(* PLC project AutBoxInterfaceOpcUa_PW02_Solution.project, Rexroth ctrlX PLC Engineering ctrlX PLC 1.20.7 *)
(* stored: creationDateTime 2025-02-11T09:05:17.5730649, modificationDateTime 2024-03-01T13:41:48 *)

(* www.hevs.ch Institut Systemes Industriels Project: Projet No: PW_01 Author: Cedric Lenoir Date: 2023 October 11 Summary: List of of components for a station of a conveyor. *)
TYPE ST_StationConveyor : STRUCT
  bButton : BOOL;
  bLed : BOOL;
  bSensor : BOOL;
END_STRUCT;
END_TYPE

(* www.hevs.ch Institut Systemes Industriels Project: Projet No: PW_01 Author: Cedric Lenoir Date: 2023 October 11 Summary: List of of components for a motor of a conveyor. *)
TYPE ST_MotorConveyor : STRUCT
  bK_ActivatePositiveDirection : BOOL;
  bK_ActivateNegativeDirection : BOOL;
END_STRUCT;
END_TYPE

(* www.hevs.ch Institut Systemes Industriels Project: Projet No: PW_02 Author: Cedric Lenoir Date: 2024 January 16 Summary: Main structure for conveyor. *)
TYPE ST_Conveyor : STRUCT
  cm01 : ST_StationConveyor;
  cm02 : ST_StationConveyor;
  cm03 : ST_StationConveyor;
  cmOut : ST_OutputConveyor;
  cmDrive : ST_MotorConveyor;
END_STRUCT;
END_TYPE

(* www.hevs.ch Institut Systemes Industriels Project: Projet No: PW_01 Author: Cedric Lenoir Date: 2024 January 14 Summary: ST_OutputConveyor extends ST_StationConveyor. *)
TYPE ST_OutputConveyor : STRUCT
  bBuzzer : BOOL;
END_STRUCT;
END_TYPE

{attribute 'qualified_only'}
VAR_GLOBAL  (* GVL_Unit *)
  myConveyor : ST_Conveyor;
END_VAR

(* www.hevs.ch Institut Systemes Industriels Project: Projet No: PW_02 Author: Cedric Lenoir Date: 2024 January 16 Summary: Main program for Pracatival Work 02. *)
PROGRAM PLC_PRG
  VAR
    diMyLoop : DINT;
    emConveyor : ST_Conveyor;
    testMode : BOOL;
    fbStationOne : FB_Station;
    fbStationTwo : FB_Station;
    fbStationThree : FB_Station;
    fbOutStation : FB_OutStation;
    fbDrive : FB_Drive;
  END_VAR

            diMyLoop := diMyLoop + 1;

//
// Manage inputs
//
// cm01
emConveyor.cm01.bButton := GVL_Abox.uaAboxInterface.uaDigitalIn.Input_0_0;
emConveyor.cm01.bSensor := GVL_Abox.uaAboxInterface.uaDigitalIn.Input_0_4;	//  UA_DigitalInput_32_Input_0_4;
// cm02
emConveyor.cm02.bButton := GVL_Abox.uaAboxInterface.uaDigitalIn.Input_0_1;
emConveyor.cm02.bSensor := GVL_Abox.uaAboxInterface.uaDigitalIn.Input_0_5;
// cm03
emConveyor.cm03.bButton := GVL_Abox.uaAboxInterface.uaDigitalIn.Input_0_2;
emConveyor.cm03.bSensor := GVL_Abox.uaAboxInterface.uaDigitalIn.Input_0_6;
// cmOut
emConveyor.cmOut.bButton := GVL_Abox.uaAboxInterface.uaDigitalIn.Input_0_3;
emConveyor.cmOut.bSensor := NOT GVL_Abox.uaAboxInterface.uaDigitalIn.Input_0_7;	// Signal inverted

// To be tested
// FC_GetInput(ioHwInterface := GVL_Abox,
//             ioPhysicalControl := emConveyor);

fbStationOne(Enable := NOT testMode, 
          ioStation := emConveyor.cm01);
fbStationTwo(Enable := NOT testMode, 
          ioStation := emConveyor.cm02);
fbStationThree(Enable := NOT testMode, 
          ioStation := emConveyor.cm03);
		  
fbOutStation(Enable := NOT testMode, 
          ioStation := emConveyor.cmOut);

		  
fbDrive(Enable := NOT testMode,
		ioDrive := emConveyor.cmDrive,
        stationOne := fbStationOne,
        stationTwo := fbStationTwo,
        stationThree := fbStationThree,
        stationOut := fbOutStation);		  

//
// Manage outputs
//
// cm01
GVL_Abox.uaAboxInterface.uaDigitalOut.Output_0_0 := emConveyor.cm01.bLed;
GVL_Abox.uaAboxInterface.uaDigitalOut.Output_0_1 := emConveyor.cm02.bLed;
GVL_Abox.uaAboxInterface.uaDigitalOut.Output_0_2 := emConveyor.cm03.bLed;
GVL_Abox.uaAboxInterface.uaDigitalOut.Output_0_3 := emConveyor.cmOut.bLed;
GVL_Abox.uaAboxInterface.uaDigitalOut.Output_0_4 := emConveyor.cmDrive.bK_ActivatePositiveDirection;
GVL_Abox.uaAboxInterface.uaDigitalOut.Output_0_5 := emConveyor.cmDrive.bK_ActivateNegativeDirection;
GVL_Abox.uaAboxInterface.uaDigitalOut.Output_0_6 := emConveyor.cmOut.bBuzzer;

// To be tested
// FC_SetOutput(ioHwInterface := GVL_Abox,
//              ioPhysicalControl := emConveyor);
          
END_PROGRAM

(* www.hevs.ch Institut Systemes Industriels Project: Projet No: PW_02 Author: Cedric Lenoir Date: 2024 January 16 Summary: Manage One station for a conveyor. *)
FUNCTION_BLOCK FB_Station
  VAR_INPUT
    Enable : BOOL;
  END_VAR
  VAR_IN_OUT
    ioStation : ST_StationConveyor;
  END_VAR
  VAR_OUTPUT
    diCounter : DINT;
    stop : BOOL;
    release : BOOL;
  END_VAR
  VAR
    rTrigIn : R_TRIG;  (* Used to count the number of inputs in station *)
    tonResetCounter : TON;  (* Reset Counte if TON for more that 2 seconds *)
  END_VAR

            IF Enable THEN
	rTrigIn(CLK := ioStation.bSensor);
	
	IF rTrigIn.Q THEN
		diCounter := diCounter + 1;
		release := FALSE;
		stop := TRUE;
	END_IF
	IF ioStation.bButton THEN
		release := TRUE;
		stop := FALSE;
	END_IF
	ioStation.bLed := stop;
	
	tonResetCounter(IN := ioStation.bButton,
					PT := T#2S);
					
	IF tonResetCounter.Q THEN
		diCounter := 0;
	END_IF
END_IF
          
END_FUNCTION_BLOCK

(* www.hevs.ch Institut Systemes Industriels Project: Projet No: PW_02 Author: Cedric Lenoir Date: 2024 January 16 Summary: Manage One station for a conveyor. *)
FUNCTION_BLOCK FB_OutStation
  VAR_INPUT
    Enable : BOOL;
  END_VAR
  VAR_IN_OUT
    ioStation : ST_OutputConveyor;
  END_VAR
  VAR_OUTPUT
    diCounter : DINT;
    stop : BOOL;
    release : BOOL;
  END_VAR
  VAR
    rTrigIn : R_TRIG;  (* Used to count the number of inputs in station *)
    tonResetCounter : TON;  (* Reset Counte if TON for more that 2 seconds *)
  END_VAR

            IF Enable THEN
	rTrigIn(CLK := ioStation.bSensor);
	
	IF rTrigIn.Q THEN
		diCounter := diCounter + 1;
		release := FALSE;
		stop := TRUE;
	END_IF
	IF ioStation.bButton THEN
		release := TRUE;
		stop := FALSE;
	END_IF
	ioStation.bLed := stop;
	
	tonResetCounter(IN := ioStation.bButton,
					PT := T#2S);
					
	IF tonResetCounter.Q THEN
		diCounter := 0;
	END_IF
	
	ioStation.bBuzzer := stop;
END_IF
          
END_FUNCTION_BLOCK

(* www.hevs.ch Institut Systemes Industriels Project: Projet No: PW_02 Author: Cedric Lenoir Date: 2024 January 16 Summary: Manage drive for motor conveyor. *)
FUNCTION_BLOCK FB_Drive
  VAR_INPUT
    Enable : BOOL;
  END_VAR
  VAR_IN_OUT
    ioDrive : ST_MotorConveyor;
    stationOne : FB_Station;
    stationTwo : FB_Station;
    stationThree : FB_Station;
    stationOut : FB_OutStation;
  END_VAR

            IF Enable THEN
	ioDrive.bK_ActivatePositiveDirection := NOT(stationOne.stop   OR 
                                                stationTwo.stop   OR
                                                stationThree.stop OR
                                                stationOut.stop);
END_IF
          
END_FUNCTION_BLOCK

(* www.hevs.ch Institut Systemes Industriels Project: Projet No: PW_01 Author: Cedric Lenoir Date: 2023 October 11 Summary: Get Physical Inputs. *)
FUNCTION FC_GetInput : BOOL
  VAR_IN_OUT
    ioHwInterface : UA_AboxInterface;
    ioPhysicalControl : ST_Conveyor;
  END_VAR

            //
// Manage inputs
//
// cm01
ioPhysicalControl.cm01.bButton := ioHwInterface.uaDigitalIn.Input_0_0;
ioPhysicalControl.cm01.bSensor := ioHwInterface.uaDigitalIn.Input_0_4;	//  UA_DigitalInput_32_Input_0_4;
// cm02
ioPhysicalControl.cm02.bButton := ioHwInterface.uaDigitalIn.Input_0_1;
ioPhysicalControl.cm02.bSensor := ioHwInterface.uaDigitalIn.Input_0_5;
// cm03
ioPhysicalControl.cm03.bButton := ioHwInterface.uaDigitalIn.Input_0_2;
ioPhysicalControl.cm03.bSensor := ioHwInterface.uaDigitalIn.Input_0_6;
// cmOut
ioPhysicalControl.cmOut.bButton := ioHwInterface.uaDigitalIn.Input_0_3;
ioPhysicalControl.cmOut.bSensor := NOT ioHwInterface.uaDigitalIn.Input_0_7;	// Signal inverted
          
END_FUNCTION

(* www.hevs.ch Institut Systemes Industriels Project: Projet No: PW_01 Author: Cedric Lenoir Date: 2024 January 11 Summary: Set Physical Inputs. *)
FUNCTION FC_SetOutput : BOOL
  VAR_IN_OUT
    ioHwInterface : UA_AboxInterface;
    ioPhysicalControl : ST_Conveyor;
  END_VAR

            ioHwInterface.uaDigitalOut.Output_0_0 := ioPhysicalControl.cm01.bLed;
ioHwInterface.uaDigitalOut.Output_0_1 := ioPhysicalControl.cm02.bLed;
ioHwInterface.uaDigitalOut.Output_0_2 := ioPhysicalControl.cm03.bLed;
ioHwInterface.uaDigitalOut.Output_0_3 := ioPhysicalControl.cmOut.bLed;
ioHwInterface.uaDigitalOut.Output_0_4 := ioPhysicalControl.cmDrive.bK_ActivatePositiveDirection;
ioHwInterface.uaDigitalOut.Output_0_5 := ioPhysicalControl.cmDrive.bK_ActivateNegativeDirection;
ioHwInterface.uaDigitalOut.Output_0_6 := ioPhysicalControl.cmOut.bBuzzer;
          
END_FUNCTION
